KUKA KRL program: flexion1.src, flexion1.dat

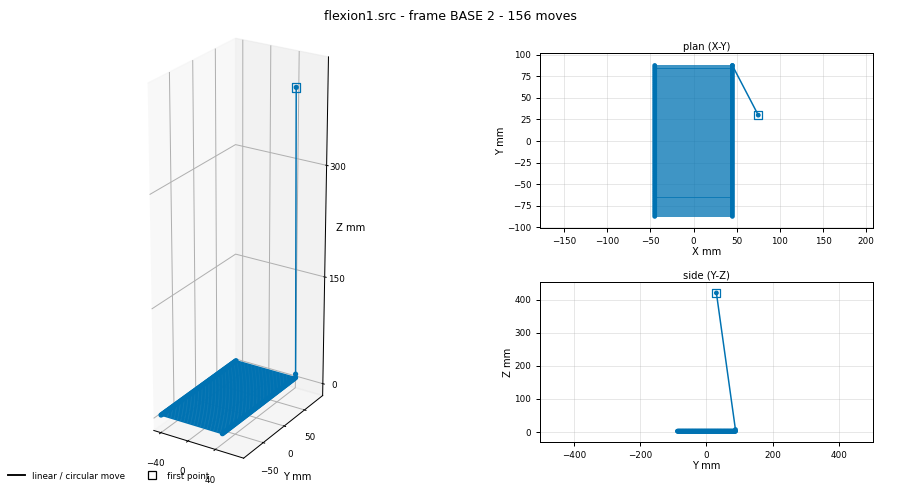
[picture p0: tool path of flexion1.src in frame BASE 2, 156 of 158 moves have a stored position in this frame; points joined in program order, loops and branches not executed]
--- flexion1.src ---
&ACCESS RVP
&PARAM TEMPLATE = C:\KRC\Roboter\Template\vorgabe
&PARAM EDITMASK = *
DEF flexion1( )
;FOLD INI;%{PE}%V3.2.0,%MKUKATPBASIS,%CINIT,%VCOMMON,%P
;FOLD BAS INI;%{E}%V3.2.0,%MKUKATPBASIS,%CINIT,%VINIT,%P
GLOBAL INTERRUPT DECL 3 WHEN $STOPMESS==TRUE DO IR_STOPM ( )
INTERRUPT ON 3
BAS (#INITMOV,0 )
;ENDFOLD (BAS INI)
;FOLD A20 INI;%{E}%V3.2.0,%MKUKATPA20,%CINIT,%VINIT,%P
IF ARC20==TRUE THEN
A20 (ARC_INI)
INTERRUPT DECL 6 WHEN $CYCFLAG[3]==FALSE DO A20(TECH_STOP2)
ENDIF
;ENDFOLD (A20 INI)
;FOLD A10 INI;%{E}%V3.2.0,%MKUKATPARC,%CINIT,%VINIT,%P
IF A10_OPTION==#ACTIVE THEN
INTERRUPT DECL 4 WHEN $CYCFLAG[2]==FALSE DO A10 (#APPL_ERROR)
INTERRUPT DECL 7 WHEN A_ARC_SWI==#ACTIVE DO A10 (#ARC_SEAM)
INTERRUPT DECL 5 WHEN A_FLY_ARC==TRUE DO A10 (#HPU_ARC)
INTERRUPT  ON 5
A10_INI ( )
ENDIF
;ENDFOLD (A10 INI)
;FOLD GRIPPER INI;%{E}%V3.2.0,%MKUKATPGRIPPER,%CINIT,%VINIT,%P
USER_GRP(0,DUMMY,DUMMY,GDEFAULT)
;ENDFOLD (GRIPPER INI)
;FOLD SPOT INI;%{E}%V3.2.0,%MKUKATPSPOT,%CINIT,%VINIT,%P
USERSPOT(#INIT)
;ENDFOLD (SPOT INI)
;FOLD TOUCHSENSE INI;%{E}%V3.2.0,%MKUKATPTS,%CINIT,%VINIT,%P
IF H70_OPTION THEN
INTERRUPT DECL 15 WHEN $MEAS_PULSE[TOUCH_I[TOUCH_ACTIVE].IN_NR] DO H70 (6,CD0 )
INTERRUPT DECL 16 WHEN $ZERO_MOVE DO H70 (7,CD0 )
INTERRUPT DECL 17 WHEN $TECHPAR_C[FG_TOUCH,8]>0.5 DO H70 (8,CD0)
H70 (1,CD0 )
ENDIF
;ENDFOLD (TOUCHSENSE INI)
;FOLD USER INI;%{E}%V3.2.0,%MKUKATPUSER,%CINIT,%VINIT,%P
;Make your modifications here
;ENDFOLD (USER INI)
;ENDFOLD (INI)
; SPEED PTP FOR AXIS
$VEL_AXIS[1] = 15
$VEL_AXIS[2] = 15
$VEL_AXIS[3] = 15
$VEL_AXIS[4] = 15
$VEL_AXIS[5] = 15
$VEL_AXIS[6] = 15
;SMOOTHNESS
$APO.CDIS = 2
;ADVANCE
$ADVANCE = 3
;SET TOOL AND BASE
$TOOL = TOOL_DATA[3]
$BASE = BASE_DATA[2]
;HOME
;FOLD PTP HOME Vel=10% DEFAULT
$BWDSTART=FALSE
$H_POS=XHOME
PDAT_ACT=PDEFAULT
FDAT_ACT=FHOME
BAS(#PTP_DAT )
BAS (#VEL_PTP,10 )
PTP XHOME
;ENDFOLD
;USER PROGRAM
;SPEED $VEL.CP
$VEL.CP=0.03
; OUT[TEMP] = 200
; OUT[vent] = 1
; OUT[RPM] = 30
; USER POSES CALLS
PTP {X 75, Y 30, Z 420, A 0, B 90, C 0}
; USER POSES CALLS
LIN {X 45.0, Y 87.5, Z 7.5, A 0, B 90, C 0} C_DIS
WAIT SEC 1
$OUT[1] = TRUE
LIN {X 45.0, Y 87.5, Z 2.5, A 0, B 90, C 0} C_DIS
LIN {X -45.0, Y 87.5, Z 2.5, A 0, B 90, C 0} C_DIS
LIN {X -45.0, Y 85.2, Z 2.5, A 0, B 90, C 0} C_DIS
LIN {X 45.0, Y 85.2, Z 2.5, A 0, B 90, C 0} C_DIS
LIN {X 45.0, Y 82.9, Z 2.5, A 0, B 90, C 0} C_DIS
LIN {X -45.0, Y 82.9, Z 2.5, A 0, B 90, C 0} C_DIS
LIN {X -45.0, Y 80.6, Z 2.5, A 0, B 90, C 0} C_DIS
LIN {X 45.0, Y 80.6, Z 2.5, A 0, B 90, C 0} C_DIS
LIN {X 45.0, Y 78.3, Z 2.5, A 0, B 90, C 0} C_DIS
LIN {X -45.0, Y 78.3, Z 2.5, A 0, B 90, C 0} C_DIS
LIN {X -45.0, Y 76.0, Z 2.5, A 0, B 90, C 0} C_DIS
LIN {X 45.0, Y 76.0, Z 2.5, A 0, B 90, C 0} C_DIS
LIN {X 45.0, Y 73.7, Z 2.5, A 0, B 90, C 0} C_DIS
LIN {X -45.0, Y 73.7, Z 2.5, A 0, B 90, C 0} C_DIS
LIN {X -45.0, Y 71.4, Z 2.5, A 0, B 90, C 0} C_DIS
LIN {X 45.0, Y 71.4, Z 2.5, A 0, B 90, C 0} C_DIS
LIN {X 45.0, Y 69.1, Z 2.5, A 0, B 90, C 0} C_DIS
LIN {X -45.0, Y 69.1, Z 2.5, A 0, B 90, C 0} C_DIS
LIN {X -45.0, Y 66.8, Z 2.5, A 0, B 90, C 0} C_DIS
LIN {X 45.0, Y 66.8, Z 2.5, A 0, B 90, C 0} C_DIS
LIN {X 45.0, Y 64.5, Z 2.5, A 0, B 90, C 0} C_DIS
LIN {X -45.0, Y 64.5, Z 2.5, A 0, B 90, C 0} C_DIS
LIN {X -45.0, Y 62.2, Z 2.5, A 0, B 90, C 0} C_DIS
LIN {X 45.0, Y 62.2, Z 2.5, A 0, B 90, C 0} C_DIS
LIN {X 45.0, Y 59.9, Z 2.5, A 0, B 90, C 0} C_DIS
LIN {X -45.0, Y 59.9, Z 2.5, A 0, B 90, C 0} C_DIS
LIN {X -45.0, Y 57.6, Z 2.5, A 0, B 90, C 0} C_DIS
LIN {X 45.0, Y 57.6, Z 2.5, A 0, B 90, C 0} C_DIS
LIN {X 45.0, Y 55.3, Z 2.5, A 0, B 90, C 0} C_DIS
LIN {X -45.0, Y 55.3, Z 2.5, A 0, B 90, C 0} C_DIS
LIN {X -45.0, Y 53.0, Z 2.5, A 0, B 90, C 0} C_DIS
LIN {X 45.0, Y 53.0, Z 2.5, A 0, B 90, C 0} C_DIS
LIN {X 45.0, Y 50.7, Z 2.5, A 0, B 90, C 0} C_DIS
LIN {X -45.0, Y 50.7, Z 2.5, A 0, B 90, C 0} C_DIS
LIN {X -45.0, Y 48.4, Z 2.5, A 0, B 90, C 0} C_DIS
LIN {X 45.0, Y 48.4, Z 2.5, A 0, B 90, C 0} C_DIS
LIN {X 45.0, Y 46.1, Z 2.5, A 0, B 90, C 0} C_DIS
LIN {X -45.0, Y 46.1, Z 2.5, A 0, B 90, C 0} C_DIS
LIN {X -45.0, Y 43.8, Z 2.5, A 0, B 90, C 0} C_DIS
LIN {X 45.0, Y 43.8, Z 2.5, A 0, B 90, C 0} C_DIS
LIN {X 45.0, Y 41.5, Z 2.5, A 0, B 90, C 0} C_DIS
LIN {X -45.0, Y 41.5, Z 2.5, A 0, B 90, C 0} C_DIS
LIN {X -45.0, Y 39.2, Z 2.5, A 0, B 90, C 0} C_DIS
LIN {X 45.0, Y 39.2, Z 2.5, A 0, B 90, C 0} C_DIS
LIN {X 45.0, Y 36.9, Z 2.5, A 0, B 90, C 0} C_DIS
LIN {X -45.0, Y 36.9, Z 2.5, A 0, B 90, C 0} C_DIS
LIN {X -45.0, Y 34.6, Z 2.5, A 0, B 90, C 0} C_DIS
LIN {X 45.0, Y 34.6, Z 2.5, A 0, B 90, C 0} C_DIS
LIN {X 45.0, Y 32.3, Z 2.5, A 0, B 90, C 0} C_DIS
LIN {X -45.0, Y 32.3, Z 2.5, A 0, B 90, C 0} C_DIS
LIN {X -45.0, Y 30.0, Z 2.5, A 0, B 90, C 0} C_DIS
LIN {X 45.0, Y 30.0, Z 2.5, A 0, B 90, C 0} C_DIS
LIN {X 45.0, Y 27.7, Z 2.5, A 0, B 90, C 0} C_DIS
LIN {X -45.0, Y 27.7, Z 2.5, A 0, B 90, C 0} C_DIS
LIN {X -45.0, Y 25.4, Z 2.5, A 0, B 90, C 0} C_DIS
LIN {X 45.0, Y 25.4, Z 2.5, A 0, B 90, C 0} C_DIS
LIN {X 45.0, Y 23.1, Z 2.5, A 0, B 90, C 0} C_DIS
LIN {X -45.0, Y 23.1, Z 2.5, A 0, B 90, C 0} C_DIS
LIN {X -45.0, Y 20.8, Z 2.5, A 0, B 90, C 0} C_DIS
LIN {X 45.0, Y 20.8, Z 2.5, A 0, B 90, C 0} C_DIS
LIN {X 45.0, Y 18.5, Z 2.5, A 0, B 90, C 0} C_DIS
LIN {X -45.0, Y 18.5, Z 2.5, A 0, B 90, C 0} C_DIS
LIN {X -45.0, Y 16.2, Z 2.5, A 0, B 90, C 0} C_DIS
LIN {X 45.0, Y 16.2, Z 2.5, A 0, B 90, C 0} C_DIS
LIN {X 45.0, Y 13.9, Z 2.5, A 0, B 90, C 0} C_DIS
LIN {X -45.0, Y 13.9, Z 2.5, A 0, B 90, C 0} C_DIS
LIN {X -45.0, Y 11.6, Z 2.5, A 0, B 90, C 0} C_DIS
LIN {X 45.0, Y 11.6, Z 2.5, A 0, B 90, C 0} C_DIS
LIN {X 45.0, Y 9.3, Z 2.5, A 0, B 90, C 0} C_DIS
LIN {X -45.0, Y 9.3, Z 2.5, A 0, B 90, C 0} C_DIS
LIN {X -45.0, Y 7.0, Z 2.5, A 0, B 90, C 0} C_DIS
LIN {X 45.0, Y 7.0, Z 2.5, A 0, B 90, C 0} C_DIS
LIN {X 45.0, Y 4.7, Z 2.5, A 0, B 90, C 0} C_DIS
LIN {X -45.0, Y 4.7, Z 2.5, A 0, B 90, C 0} C_DIS
LIN {X -45.0, Y 2.4, Z 2.5, A 0, B 90, C 0} C_DIS
LIN {X 45.0, Y 2.4, Z 2.5, A 0, B 90, C 0} C_DIS
LIN {X 45.0, Y 0.1, Z 2.5, A 0, B 90, C 0} C_DIS
LIN {X -45.0, Y 0.1, Z 2.5, A 0, B 90, C 0} C_DIS
LIN {X -45.0, Y -2.2, Z 2.5, A 0, B 90, C 0} C_DIS
LIN {X 45.0, Y -2.2, Z 2.5, A 0, B 90, C 0} C_DIS
LIN {X 45.0, Y -4.5, Z 2.5, A 0, B 90, C 0} C_DIS
LIN {X -45.0, Y -4.5, Z 2.5, A 0, B 90, C 0} C_DIS
LIN {X -45.0, Y -6.8, Z 2.5, A 0, B 90, C 0} C_DIS
LIN {X 45.0, Y -6.8, Z 2.5, A 0, B 90, C 0} C_DIS
LIN {X 45.0, Y -9.1, Z 2.5, A 0, B 90, C 0} C_DIS
LIN {X -45.0, Y -9.1, Z 2.5, A 0, B 90, C 0} C_DIS
LIN {X -45.0, Y -11.4, Z 2.5, A 0, B 90, C 0} C_DIS
LIN {X 45.0, Y -11.4, Z 2.5, A 0, B 90, C 0} C_DIS
LIN {X 45.0, Y -13.7, Z 2.5, A 0, B 90, C 0} C_DIS
LIN {X -45.0, Y -13.7, Z 2.5, A 0, B 90, C 0} C_DIS
LIN {X -45.0, Y -16.0, Z 2.5, A 0, B 90, C 0} C_DIS
LIN {X 45.0, Y -16.0, Z 2.5, A 0, B 90, C 0} C_DIS
LIN {X 45.0, Y -18.3, Z 2.5, A 0, B 90, C 0} C_DIS
LIN {X -45.0, Y -18.3, Z 2.5, A 0, B 90, C 0} C_DIS
LIN {X -45.0, Y -20.6, Z 2.5, A 0, B 90, C 0} C_DIS
LIN {X 45.0, Y -20.6, Z 2.5, A 0, B 90, C 0} C_DIS
LIN {X 45.0, Y -22.9, Z 2.5, A 0, B 90, C 0} C_DIS
LIN {X -45.0, Y -22.9, Z 2.5, A 0, B 90, C 0} C_DIS
LIN {X -45.0, Y -25.2, Z 2.5, A 0, B 90, C 0} C_DIS
LIN {X 45.0, Y -25.2, Z 2.5, A 0, B 90, C 0} C_DIS
LIN {X 45.0, Y -27.5, Z 2.5, A 0, B 90, C 0} C_DIS
LIN {X -45.0, Y -27.5, Z 2.5, A 0, B 90, C 0} C_DIS
LIN {X -45.0, Y -29.8, Z 2.5, A 0, B 90, C 0} C_DIS
LIN {X 45.0, Y -29.8, Z 2.5, A 0, B 90, C 0} C_DIS
LIN {X 45.0, Y -32.1, Z 2.5, A 0, B 90, C 0} C_DIS
LIN {X -45.0, Y -32.1, Z 2.5, A 0, B 90, C 0} C_DIS
LIN {X -45.0, Y -34.4, Z 2.5, A 0, B 90, C 0} C_DIS
LIN {X 45.0, Y -34.4, Z 2.5, A 0, B 90, C 0} C_DIS
LIN {X 45.0, Y -36.7, Z 2.5, A 0, B 90, C 0} C_DIS
LIN {X -45.0, Y -36.7, Z 2.5, A 0, B 90, C 0} C_DIS
LIN {X -45.0, Y -39.0, Z 2.5, A 0, B 90, C 0} C_DIS
LIN {X 45.0, Y -39.0, Z 2.5, A 0, B 90, C 0} C_DIS
LIN {X 45.0, Y -41.3, Z 2.5, A 0, B 90, C 0} C_DIS
LIN {X -45.0, Y -41.3, Z 2.5, A 0, B 90, C 0} C_DIS
LIN {X -45.0, Y -43.6, Z 2.5, A 0, B 90, C 0} C_DIS
LIN {X 45.0, Y -43.6, Z 2.5, A 0, B 90, C 0} C_DIS
LIN {X 45.0, Y -45.9, Z 2.5, A 0, B 90, C 0} C_DIS
LIN {X -45.0, Y -45.9, Z 2.5, A 0, B 90, C 0} C_DIS
LIN {X -45.0, Y -48.2, Z 2.5, A 0, B 90, C 0} C_DIS
LIN {X 45.0, Y -48.2, Z 2.5, A 0, B 90, C 0} C_DIS
LIN {X 45.0, Y -50.5, Z 2.5, A 0, B 90, C 0} C_DIS
LIN {X -45.0, Y -50.5, Z 2.5, A 0, B 90, C 0} C_DIS
LIN {X -45.0, Y -52.8, Z 2.5, A 0, B 90, C 0} C_DIS
LIN {X 45.0, Y -52.8, Z 2.5, A 0, B 90, C 0} C_DIS
LIN {X 45.0, Y -55.1, Z 2.5, A 0, B 90, C 0} C_DIS
LIN {X -45.0, Y -55.1, Z 2.5, A 0, B 90, C 0} C_DIS
LIN {X -45.0, Y -57.4, Z 2.5, A 0, B 90, C 0} C_DIS
LIN {X 45.0, Y -57.4, Z 2.5, A 0, B 90, C 0} C_DIS
LIN {X 45.0, Y -59.7, Z 2.5, A 0, B 90, C 0} C_DIS
LIN {X -45.0, Y -59.7, Z 2.5, A 0, B 90, C 0} C_DIS
LIN {X -45.0, Y -62.0, Z 2.5, A 0, B 90, C 0} C_DIS
LIN {X 45.0, Y -62.0, Z 2.5, A 0, B 90, C 0} C_DIS
LIN {X 45.0, Y -64.3, Z 2.5, A 0, B 90, C 0} C_DIS
LIN {X -45.0, Y -64.3, Z 2.5, A 0, B 90, C 0} C_DIS
LIN {X -45.0, Y -66.6, Z 2.5, A 0, B 90, C 0} C_DIS
LIN {X 45.0, Y -66.6, Z 2.5, A 0, B 90, C 0} C_DIS
LIN {X 45.0, Y -68.9, Z 2.5, A 0, B 90, C 0} C_DIS
LIN {X -45.0, Y -68.9, Z 2.5, A 0, B 90, C 0} C_DIS
LIN {X -45.0, Y -71.2, Z 2.5, A 0, B 90, C 0} C_DIS
LIN {X 45.0, Y -71.2, Z 2.5, A 0, B 90, C 0} C_DIS
LIN {X 45.0, Y -73.5, Z 2.5, A 0, B 90, C 0} C_DIS
LIN {X -45.0, Y -73.5, Z 2.5, A 0, B 90, C 0} C_DIS
LIN {X -45.0, Y -75.8, Z 2.5, A 0, B 90, C 0} C_DIS
LIN {X 45.0, Y -75.8, Z 2.5, A 0, B 90, C 0} C_DIS
LIN {X 45.0, Y -78.1, Z 2.5, A 0, B 90, C 0} C_DIS
LIN {X -45.0, Y -78.1, Z 2.5, A 0, B 90, C 0} C_DIS
LIN {X -45.0, Y -80.4, Z 2.5, A 0, B 90, C 0} C_DIS
LIN {X 45.0, Y -80.4, Z 2.5, A 0, B 90, C 0} C_DIS
LIN {X 45.0, Y -82.7, Z 2.5, A 0, B 90, C 0} C_DIS
LIN {X -45.0, Y -82.7, Z 2.5, A 0, B 90, C 0} C_DIS
LIN {X -45.0, Y -85.0, Z 2.5, A 0, B 90, C 0} C_DIS
LIN {X 45.0, Y -85.0, Z 2.5, A 0, B 90, C 0} C_DIS
LIN {X 45.0, Y -87.3, Z 2.5, A 0, B 90, C 0} C_DIS
LIN {X -45.0, Y -87.3, Z 2.5, A 0, B 90, C 0} C_DIS
$OUT[1] = FALSE

;Wait for
; END POSITION FOR
;END USER CODE
;HOME
;FOLD PTP HOME Vel=10% DEFAULT
$BWDSTART=FALSE
$H_POS=XHOME
PDAT_ACT=PDEFAULT
FDAT_ACT=FHOME
BAS(#PTP_DAT )
BAS (#VEL_PTP,10 )
PTP XHOME
;ENDFOLD
END

--- flexion1.dat ---
DEFDAT flexion1()
ENDDAT
